// TIA Portal V17 export
// export: Created 2025-03-05T07:59:29.2018149Z, ExportSetting WithDefaults, DisplayName Totally Integrated Automation Portal, DisplayVersion V17 Update 8, DisplayName TIA Portal Openness, DisplayVersion V17 Update 8, DisplayName TIA Portal Version Control Interface, DisplayVersion V17, DisplayName SINAMICS Startdrive Advanced, DisplayVersion V17 SP2, DisplayName SINAMICS Startdrive G110M, G120, G120C, G120D, G120P, G115D, DisplayVersion V17 SP2, DisplayName SINAMICS Startdrive G130, G150, S120, S150, SINAMICS MV, S210, DisplayVersion V17 SP2, DisplayName STEP 7 Professional, DisplayVersion V17 Update 8, DisplayName SINUMERIK ONE STEP 7 Toolbox, DisplayVersion V17 Update 12, DisplayName SINUMERIK 840D sl STEP 7 Toolbox, DisplayVersion V17 Update 12, DisplayName STEP 7 Safety, DisplayVersion V17 Update 6, DisplayName WinCC Advanced, DisplayVersion V17 Update 8
FUNCTION_BLOCK "FB301_CHANNEL_READ_AXES_POSITIONS"   // FB301, LAD
{ S7_Optimized_Access := 'FALSE' }
AUTHOR : ETXETAR
VERSION : 1.0
// stored: AutoNumber false, IsIECCheckEnabled false, SetENOAutomatically false, UDAEnableTagReadback false
   VAR_INPUT
      NUMBER_AXES_GROUP_1 : Int;   // MAX. VALUE 8 / NUMBER AXES GROUP 1, MAX=8
      NUMBER_AXES_GROUP_2 : Int;   // MAX. VALUE 7 / NUMBER AXES GROUP 2, MAX=8
      NUMBER_AXES_GROUP_3 : Int;   // MAX. VALUE 7 / NUMBER AXES GROUP 3, MAX=4
   END_VAR
   VAR_OUTPUT
      ALARM : Bool;   // ALARM
      AXIS_POSITION_1 : DWord;   // AXIS POSITION 1
      AXIS_POSITION_2 : DWord;   // AXIS POSITION 2
      AXIS_POSITION_3 : DWord;   // AXIS POSITION 3
      AXIS_POSITION_4 : DWord;   // AXIS POSITION 4
      AXIS_POSITION_5 : DWord;   // AXIS POSITION 5
      AXIS_POSITION_6 : DWord;   // AXIS POSITION 6
      AXIS_POSITION_7 : DWord;   // AXIS POSITION 7
      AXIS_POSITION_8 : DWord;   // AXIS POSITION 8
      AXIS_POSITION_9 : DWord;   // AXIS POSITION 9
      AXIS_POSITION_10 : DWord;   // AXIS POSITION 10
      AXIS_POSITION_11 : DWord;   // AXIS POSITION 11
      AXIS_POSITION_12 : DWord;   // AXIS POSITION 12
      AXIS_POSITION_13 : DWord;   // AXIS POSITION 13
      AXIS_POSITION_14 : DWord;   // AXIS POSITION 14
      AXIS_POSITION_15 : DWord;   // AXIS POSITION 15
      AXIS_POSITION_16 : DWord;   // AXIS POSITION 16
      AXIS_POSITION_17 : DWord;   // AXIS POSITION 17
      AXIS_POSITION_18 : DWord;   // AXIS POSITION 18
      AXIS_POSITION_19 : DWord;   // AXIS POSITION 19
      AXIS_POSITION_20 : DWord;   // AXIS POSITION 20
   END_VAR
   VAR DB_SPECIFIC
      readDB { S7_SetPoint := 'True'} : "READ_AXES_POSITIONS_CH";
   END_VAR
   VAR
      FB2_Instance_1 { S7_SetPoint := 'True'} : "LBP_ReadVar";
      FB2_Instance_2 { S7_SetPoint := 'True'} : "LBP_ReadVar";
      FB2_Instance_3 { S7_SetPoint := 'True'} : "LBP_ReadVar";
   END_VAR
   VAR DB_SPECIFIC
      FAULT_COUNTER { S7_SetPoint := 'True'} : CTU_INT;
   END_VAR
   VAR_TEMP
      DB_NUMBER : DInt;   // DB NUMBER FOR ALARM AND HELP DECODING
      CHANNEL : UInt;   // CHANNEL NUMBER MAX. NUMBER=10
      FAULT : Bool;   // FAULT
      COUNT_ERRORS : Int;   // COUNT_ERRORS
   END_VAR
   VAR_TEMP   // added for the SCL form of the ladder/FBD networks
      _w1 : Bool;
   END_VAR
BEGIN

NETWORK
TITLE = READ INSTANCE DB
      L     DINO;
      +     10#800000;
      T     #DB_NUMBER;
      L     DINO;
      L     10#300;
      -I;
      T     #CHANNEL;



REGION Network 2: FAULT / CHANNELS READING FAULT
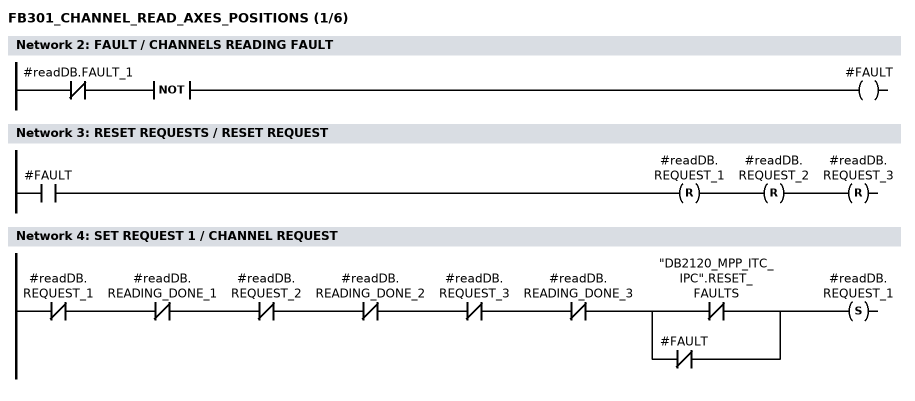
   RUNG wire#powerrail
      I_Contact( #readDB.FAULT_1 )
      Not()
      Coil( #FAULT )
   END_RUNG
   // the same network as SCL:
   #FAULT := NOT (NOT #readDB.FAULT_1);
END_REGION

REGION Network 3: RESET REQUESTS / RESET REQUEST
   RUNG wire#powerrail
      Contact( #FAULT )
      R_Coil( #readDB.REQUEST_1 )
      R_Coil( #readDB.REQUEST_2 )
      R_Coil( #readDB.REQUEST_3 )
   END_RUNG
   // the same network as SCL:
   IF #FAULT THEN
       #readDB.REQUEST_1 := FALSE;
       #readDB.REQUEST_2 := FALSE;
       #readDB.REQUEST_3 := FALSE;
   END_IF;
END_REGION

REGION Network 4: SET REQUEST 1 / CHANNEL REQUEST
   RUNG wire#powerrail
      I_Contact( #readDB.REQUEST_1 )
      I_Contact( #readDB.READING_DONE_1 )
      I_Contact( #readDB.REQUEST_2 )
      I_Contact( #readDB.READING_DONE_2 )
      I_Contact( #readDB.REQUEST_3 )
      I_Contact( #readDB.READING_DONE_3 )
      wire#w1
      I_Contact( "DB2120_MPP_ITC_IPC".RESET_FAULTS )
      wire#w2
      S_Coil( #readDB.REQUEST_1 )
   END_RUNG
   RUNG wire#w1
      I_Contact( #FAULT )
   END_RUNG wire#w2
   // the same network as SCL:
   IF NOT #readDB.REQUEST_1 AND NOT #readDB.READING_DONE_1 AND NOT #readDB.REQUEST_2 AND NOT #readDB.READING_DONE_2 AND NOT #readDB.REQUEST_3 AND NOT #readDB.READING_DONE_3 AND (NOT "DB2120_MPP_ITC_IPC".RESET_FAULTS OR NOT #FAULT) THEN
       #readDB.REQUEST_1 := TRUE;
   END_IF;
END_REGION

REGION Network 5: CALL FB2 GROUP 1 / READ AXES POSITIONS CHANNEL
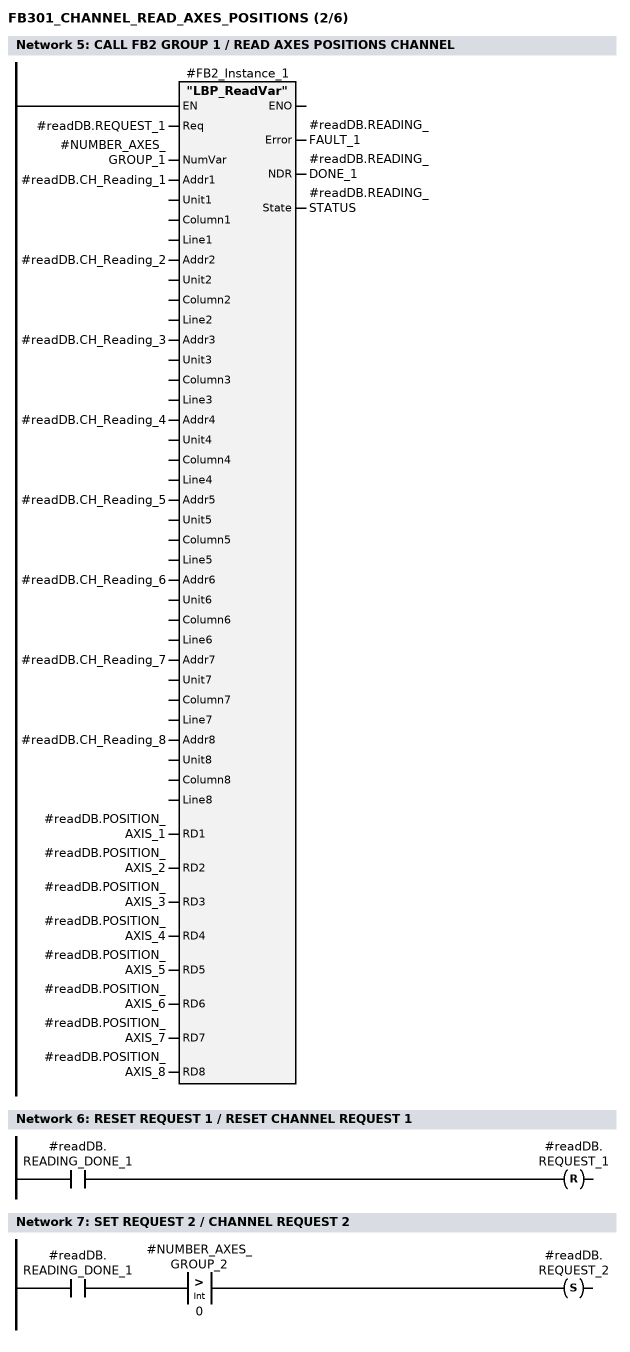
   RUNG wire#powerrail
      #FB2_Instance_1(Req := #readDB.REQUEST_1, NumVar := #NUMBER_AXES_GROUP_1, Addr1 := #readDB.CH_Reading_1, Unit1 :=, Column1 :=, Line1 :=, Addr2 := #readDB.CH_Reading_2, Unit2 :=, Column2 :=, Line2 :=, Addr3 := #readDB.CH_Reading_3, Unit3 :=, Column3 :=, Line3 :=, Addr4 := #readDB.CH_Reading_4, Unit4 :=, Column4 :=, Line4 :=, Addr5 := #readDB.CH_Reading_5, Unit5 :=, Column5 :=, Line5 :=, Addr6 := #readDB.CH_Reading_6, Unit6 :=, Column6 :=, Line6 :=, Addr7 := #readDB.CH_Reading_7, Unit7 :=, Column7 :=, Line7 :=, Addr8 := #readDB.CH_Reading_8, Unit8 :=, Column8 :=, Line8 :=, RD1 := #readDB.POSITION_AXIS_1, RD2 := #readDB.POSITION_AXIS_2, RD3 := #readDB.POSITION_AXIS_3, RD4 := #readDB.POSITION_AXIS_4, RD5 := #readDB.POSITION_AXIS_5, RD6 := #readDB.POSITION_AXIS_6, RD7 := #readDB.POSITION_AXIS_7, RD8 := #readDB.POSITION_AXIS_8, Error => #readDB.READING_FAULT_1, NDR => #readDB.READING_DONE_1, State => #readDB.READING_STATUS)
   END_RUNG
   // the same network as SCL:
   #FB2_Instance_1(Req := #readDB.REQUEST_1,   // "LBP_ReadVar"
                   NumVar := #NUMBER_AXES_GROUP_1,
                   Addr1 := #readDB.CH_Reading_1,
                   Addr2 := #readDB.CH_Reading_2,
                   Addr3 := #readDB.CH_Reading_3,
                   Addr4 := #readDB.CH_Reading_4,
                   Addr5 := #readDB.CH_Reading_5,
                   Addr6 := #readDB.CH_Reading_6,
                   Addr7 := #readDB.CH_Reading_7,
                   Addr8 := #readDB.CH_Reading_8,
                   RD1 := #readDB.POSITION_AXIS_1,
                   RD2 := #readDB.POSITION_AXIS_2,
                   RD3 := #readDB.POSITION_AXIS_3,
                   RD4 := #readDB.POSITION_AXIS_4,
                   RD5 := #readDB.POSITION_AXIS_5,
                   RD6 := #readDB.POSITION_AXIS_6,
                   RD7 := #readDB.POSITION_AXIS_7,
                   RD8 := #readDB.POSITION_AXIS_8,
                   Error => #readDB.READING_FAULT_1,
                   NDR => #readDB.READING_DONE_1,
                   State => #readDB.READING_STATUS);
END_REGION

REGION Network 6: RESET REQUEST 1 / RESET CHANNEL REQUEST 1
   RUNG wire#powerrail
      Contact( #readDB.READING_DONE_1 )
      R_Coil( #readDB.REQUEST_1 )
   END_RUNG
   // the same network as SCL:
   IF #readDB.READING_DONE_1 THEN #readDB.REQUEST_1 := FALSE; END_IF;
END_REGION

REGION Network 7: SET REQUEST 2 / CHANNEL REQUEST 2
   RUNG wire#powerrail
      Contact( #readDB.READING_DONE_1 )
      { S7_Templates := "SrcType := Int" } GT_Contact(in1 := #NUMBER_AXES_GROUP_2, in2 := 0)
      S_Coil( #readDB.REQUEST_2 )
   END_RUNG
   // the same network as SCL:
   IF #readDB.READING_DONE_1 AND (#NUMBER_AXES_GROUP_2 > 0) THEN #readDB.REQUEST_2 := TRUE; END_IF;
END_REGION

REGION Network 8: CALL FB2 GROUP 2 / READ AXES POSITIONS CHANNEL
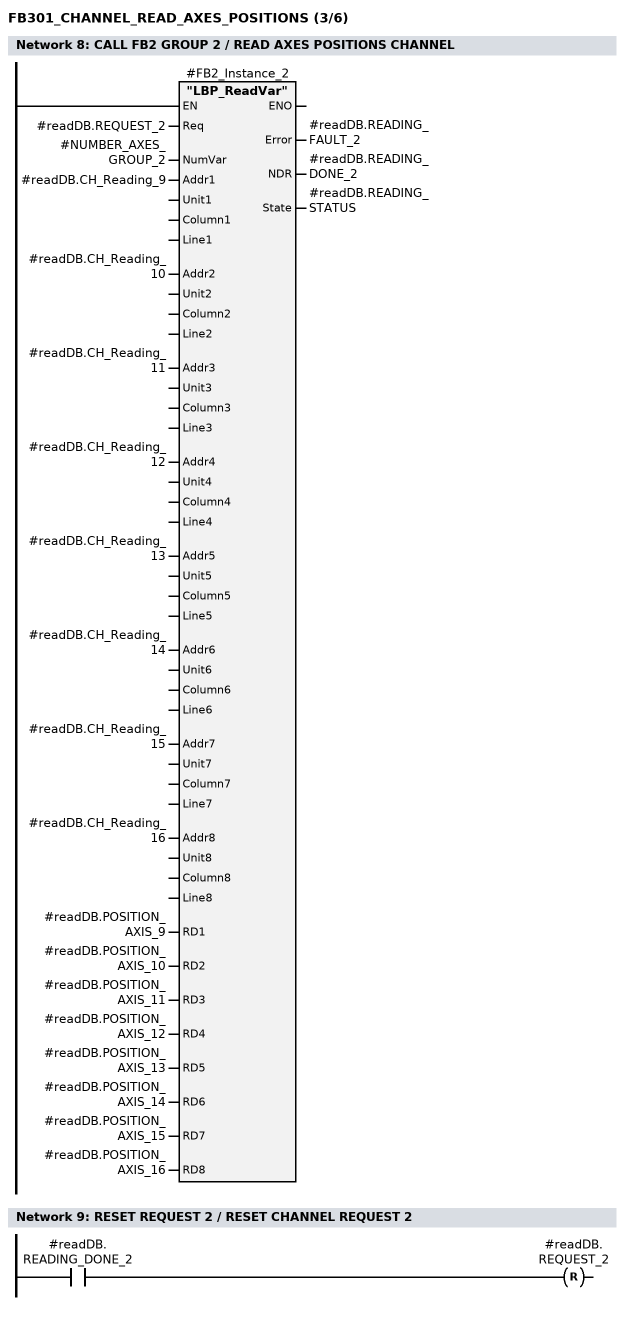
   RUNG wire#powerrail
      #FB2_Instance_2(Req := #readDB.REQUEST_2, NumVar := #NUMBER_AXES_GROUP_2, Addr1 := #readDB.CH_Reading_9, Unit1 :=, Column1 :=, Line1 :=, Addr2 := #readDB.CH_Reading_10, Unit2 :=, Column2 :=, Line2 :=, Addr3 := #readDB.CH_Reading_11, Unit3 :=, Column3 :=, Line3 :=, Addr4 := #readDB.CH_Reading_12, Unit4 :=, Column4 :=, Line4 :=, Addr5 := #readDB.CH_Reading_13, Unit5 :=, Column5 :=, Line5 :=, Addr6 := #readDB.CH_Reading_14, Unit6 :=, Column6 :=, Line6 :=, Addr7 := #readDB.CH_Reading_15, Unit7 :=, Column7 :=, Line7 :=, Addr8 := #readDB.CH_Reading_16, Unit8 :=, Column8 :=, Line8 :=, RD1 := #readDB.POSITION_AXIS_9, RD2 := #readDB.POSITION_AXIS_10, RD3 := #readDB.POSITION_AXIS_11, RD4 := #readDB.POSITION_AXIS_12, RD5 := #readDB.POSITION_AXIS_13, RD6 := #readDB.POSITION_AXIS_14, RD7 := #readDB.POSITION_AXIS_15, RD8 := #readDB.POSITION_AXIS_16, Error => #readDB.READING_FAULT_2, NDR => #readDB.READING_DONE_2, State => #readDB.READING_STATUS)
   END_RUNG
   // the same network as SCL:
   #FB2_Instance_2(Req := #readDB.REQUEST_2,   // "LBP_ReadVar"
                   NumVar := #NUMBER_AXES_GROUP_2,
                   Addr1 := #readDB.CH_Reading_9,
                   Addr2 := #readDB.CH_Reading_10,
                   Addr3 := #readDB.CH_Reading_11,
                   Addr4 := #readDB.CH_Reading_12,
                   Addr5 := #readDB.CH_Reading_13,
                   Addr6 := #readDB.CH_Reading_14,
                   Addr7 := #readDB.CH_Reading_15,
                   Addr8 := #readDB.CH_Reading_16,
                   RD1 := #readDB.POSITION_AXIS_9,
                   RD2 := #readDB.POSITION_AXIS_10,
                   RD3 := #readDB.POSITION_AXIS_11,
                   RD4 := #readDB.POSITION_AXIS_12,
                   RD5 := #readDB.POSITION_AXIS_13,
                   RD6 := #readDB.POSITION_AXIS_14,
                   RD7 := #readDB.POSITION_AXIS_15,
                   RD8 := #readDB.POSITION_AXIS_16,
                   Error => #readDB.READING_FAULT_2,
                   NDR => #readDB.READING_DONE_2,
                   State => #readDB.READING_STATUS);
END_REGION

REGION Network 9: RESET REQUEST 2 / RESET CHANNEL REQUEST 2
   RUNG wire#powerrail
      Contact( #readDB.READING_DONE_2 )
      R_Coil( #readDB.REQUEST_2 )
   END_RUNG
   // the same network as SCL:
   IF #readDB.READING_DONE_2 THEN #readDB.REQUEST_2 := FALSE; END_IF;
END_REGION

REGION Network 10: SET REQUEST 3 / RESET CHANNEL REQUEST 2
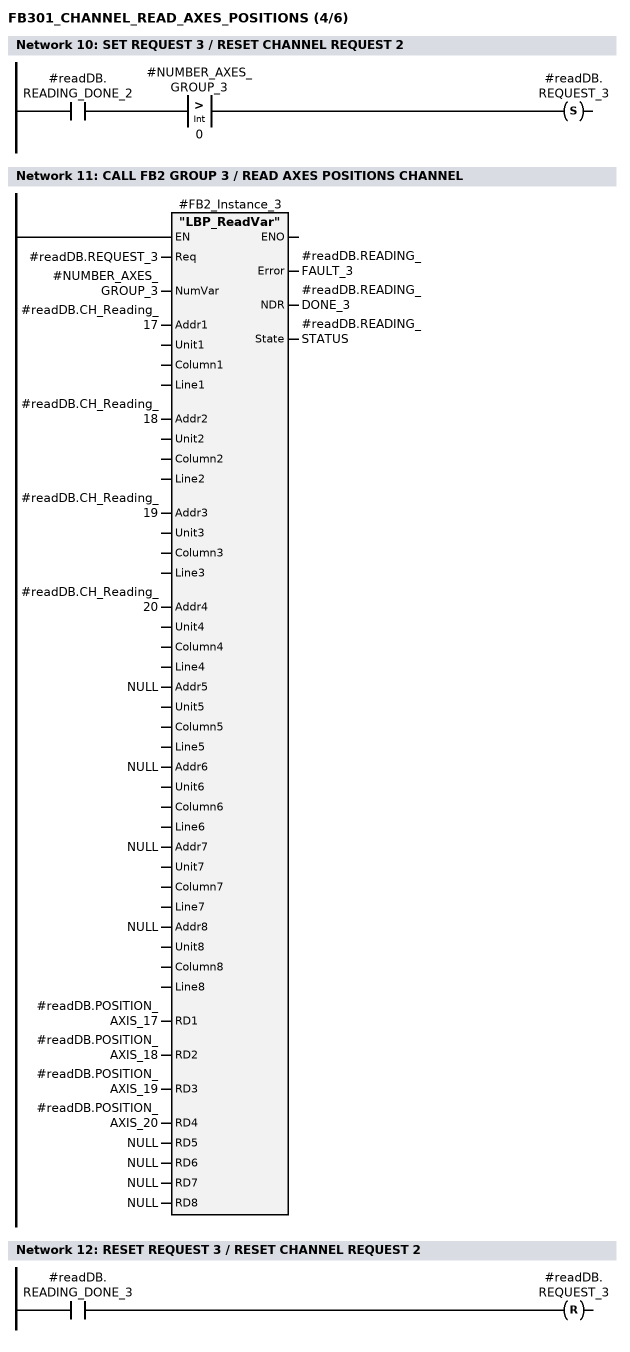
   RUNG wire#powerrail
      Contact( #readDB.READING_DONE_2 )
      { S7_Templates := "SrcType := Int" } GT_Contact(in1 := #NUMBER_AXES_GROUP_3, in2 := 0)
      S_Coil( #readDB.REQUEST_3 )
   END_RUNG
   // the same network as SCL:
   IF #readDB.READING_DONE_2 AND (#NUMBER_AXES_GROUP_3 > 0) THEN #readDB.REQUEST_3 := TRUE; END_IF;
END_REGION

REGION Network 11: CALL FB2 GROUP 3 / READ AXES POSITIONS CHANNEL
   RUNG wire#powerrail
      #FB2_Instance_3(Req := #readDB.REQUEST_3, NumVar := #NUMBER_AXES_GROUP_3, Addr1 := #readDB.CH_Reading_17, Unit1 :=, Column1 :=, Line1 :=, Addr2 := #readDB.CH_Reading_18, Unit2 :=, Column2 :=, Line2 :=, Addr3 := #readDB.CH_Reading_19, Unit3 :=, Column3 :=, Line3 :=, Addr4 := #readDB.CH_Reading_20, Unit4 :=, Column4 :=, Line4 :=, Addr5 := NULL, Unit5 :=, Column5 :=, Line5 :=, Addr6 := NULL, Unit6 :=, Column6 :=, Line6 :=, Addr7 := NULL, Unit7 :=, Column7 :=, Line7 :=, Addr8 := NULL, Unit8 :=, Column8 :=, Line8 :=, RD1 := #readDB.POSITION_AXIS_17, RD2 := #readDB.POSITION_AXIS_18, RD3 := #readDB.POSITION_AXIS_19, RD4 := #readDB.POSITION_AXIS_20, RD5 := NULL, RD6 := NULL, RD7 := NULL, RD8 := NULL, Error => #readDB.READING_FAULT_3, NDR => #readDB.READING_DONE_3, State => #readDB.READING_STATUS)
   END_RUNG
   // the same network as SCL:
   #FB2_Instance_3(Req := #readDB.REQUEST_3,   // "LBP_ReadVar"
                   NumVar := #NUMBER_AXES_GROUP_3,
                   Addr1 := #readDB.CH_Reading_17,
                   Addr2 := #readDB.CH_Reading_18,
                   Addr3 := #readDB.CH_Reading_19,
                   Addr4 := #readDB.CH_Reading_20,
                   Addr5 := NULL,
                   Addr6 := NULL,
                   Addr7 := NULL,
                   Addr8 := NULL,
                   RD1 := #readDB.POSITION_AXIS_17,
                   RD2 := #readDB.POSITION_AXIS_18,
                   RD3 := #readDB.POSITION_AXIS_19,
                   RD4 := #readDB.POSITION_AXIS_20,
                   RD5 := NULL,
                   RD6 := NULL,
                   RD7 := NULL,
                   RD8 := NULL,
                   Error => #readDB.READING_FAULT_3,
                   NDR => #readDB.READING_DONE_3,
                   State => #readDB.READING_STATUS);
END_REGION

REGION Network 12: RESET REQUEST 3 / RESET CHANNEL REQUEST 2
   RUNG wire#powerrail
      Contact( #readDB.READING_DONE_3 )
      R_Coil( #readDB.REQUEST_3 )
   END_RUNG
   // the same network as SCL:
   IF #readDB.READING_DONE_3 THEN #readDB.REQUEST_3 := FALSE; END_IF;
END_REGION

REGION Network 13: MOVE POSITIONS / AXES POSITIONS
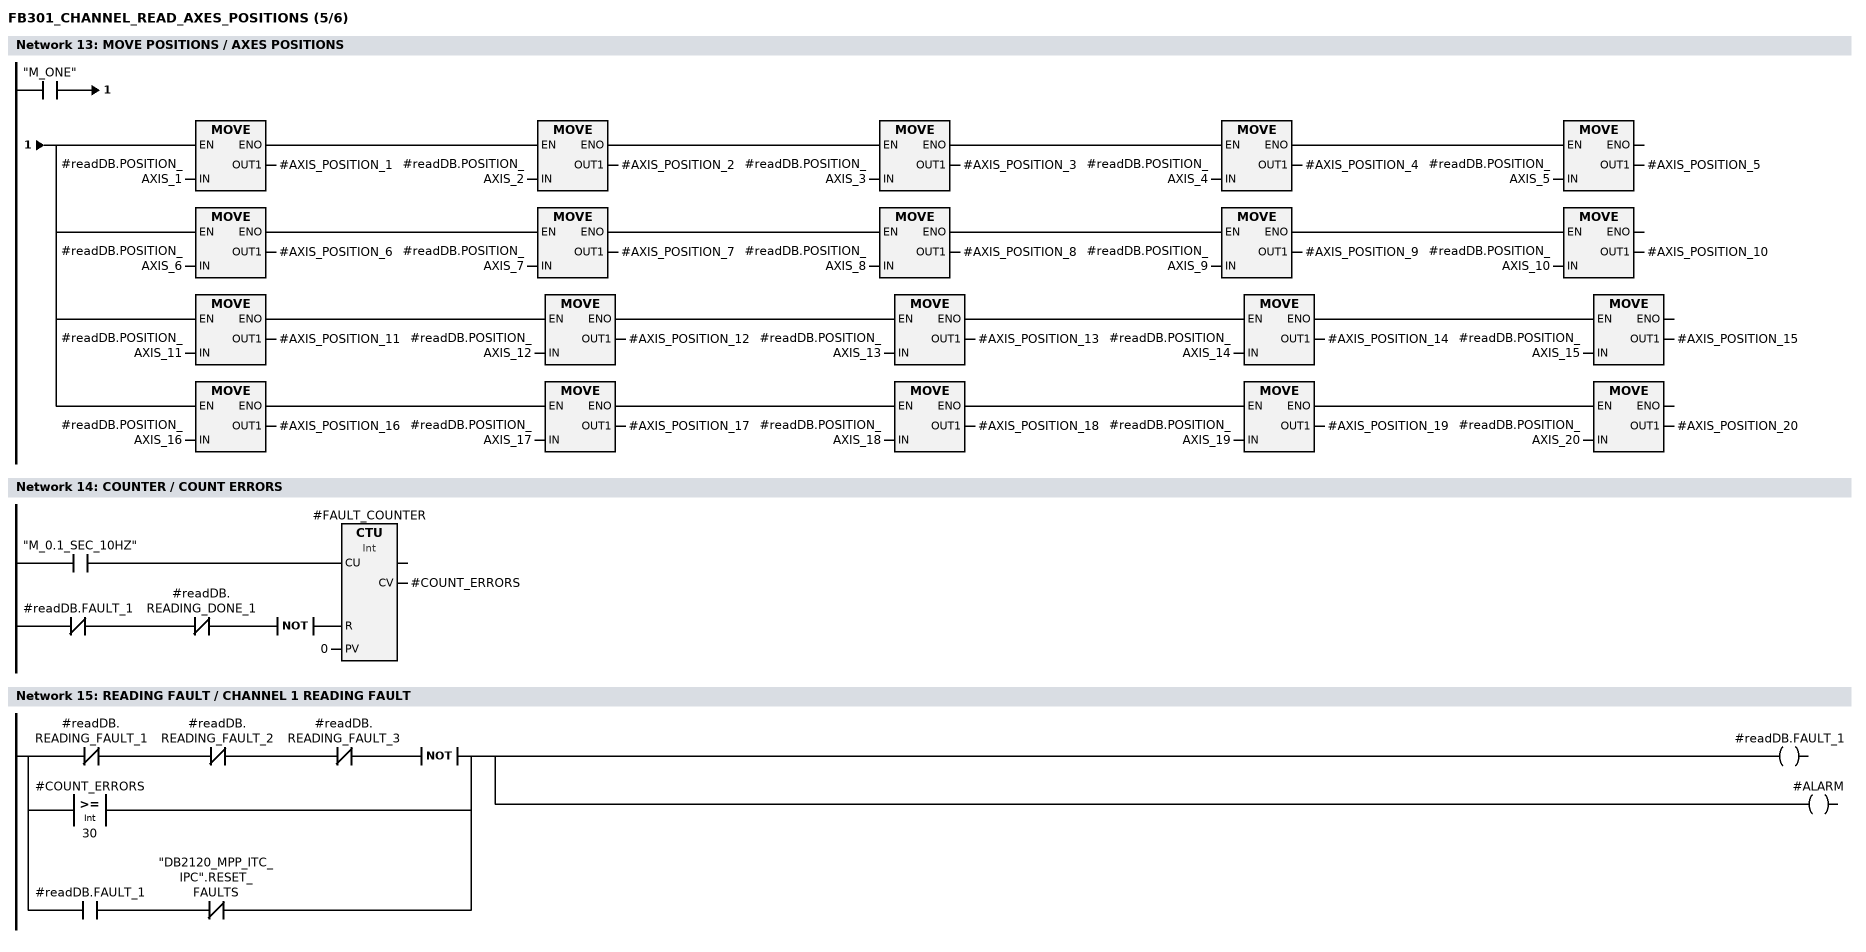
   RUNG wire#powerrail
      Contact( "M_ONE" )
      wire#w1
      { S7_GenerateENO := "TRUE" } Move(in := #readDB.POSITION_AXIS_1, out1 => #AXIS_POSITION_1)
      { S7_GenerateENO := "TRUE" } Move(in := #readDB.POSITION_AXIS_2, out1 => #AXIS_POSITION_2)
      { S7_GenerateENO := "TRUE" } Move(in := #readDB.POSITION_AXIS_3, out1 => #AXIS_POSITION_3)
      { S7_GenerateENO := "TRUE" } Move(in := #readDB.POSITION_AXIS_4, out1 => #AXIS_POSITION_4)
      { S7_GenerateENO := "TRUE" } Move(in := #readDB.POSITION_AXIS_5, out1 => #AXIS_POSITION_5)
   END_RUNG
   RUNG wire#w1
      { S7_GenerateENO := "TRUE" } Move(in := #readDB.POSITION_AXIS_6, out1 => #AXIS_POSITION_6)
      { S7_GenerateENO := "TRUE" } Move(in := #readDB.POSITION_AXIS_7, out1 => #AXIS_POSITION_7)
      { S7_GenerateENO := "TRUE" } Move(in := #readDB.POSITION_AXIS_8, out1 => #AXIS_POSITION_8)
      { S7_GenerateENO := "TRUE" } Move(in := #readDB.POSITION_AXIS_9, out1 => #AXIS_POSITION_9)
      { S7_GenerateENO := "TRUE" } Move(in := #readDB.POSITION_AXIS_10, out1 => #AXIS_POSITION_10)
   END_RUNG
   RUNG wire#w1
      { S7_GenerateENO := "TRUE" } Move(in := #readDB.POSITION_AXIS_11, out1 => #AXIS_POSITION_11)
      { S7_GenerateENO := "TRUE" } Move(in := #readDB.POSITION_AXIS_12, out1 => #AXIS_POSITION_12)
      { S7_GenerateENO := "TRUE" } Move(in := #readDB.POSITION_AXIS_13, out1 => #AXIS_POSITION_13)
      { S7_GenerateENO := "TRUE" } Move(in := #readDB.POSITION_AXIS_14, out1 => #AXIS_POSITION_14)
      { S7_GenerateENO := "TRUE" } Move(in := #readDB.POSITION_AXIS_15, out1 => #AXIS_POSITION_15)
   END_RUNG
   RUNG wire#w1
      { S7_GenerateENO := "TRUE" } Move(in := #readDB.POSITION_AXIS_16, out1 => #AXIS_POSITION_16)
      { S7_GenerateENO := "TRUE" } Move(in := #readDB.POSITION_AXIS_17, out1 => #AXIS_POSITION_17)
      { S7_GenerateENO := "TRUE" } Move(in := #readDB.POSITION_AXIS_18, out1 => #AXIS_POSITION_18)
      { S7_GenerateENO := "TRUE" } Move(in := #readDB.POSITION_AXIS_19, out1 => #AXIS_POSITION_19)
      { S7_GenerateENO := "TRUE" } Move(in := #readDB.POSITION_AXIS_20, out1 => #AXIS_POSITION_20)
   END_RUNG
   // the same network as SCL:
   // ENO of a box is taken as its EN; it also drops when the box reports an error
   IF "M_ONE" THEN
       #AXIS_POSITION_1 := #readDB.POSITION_AXIS_1;
       #AXIS_POSITION_2 := #readDB.POSITION_AXIS_2;
       #AXIS_POSITION_3 := #readDB.POSITION_AXIS_3;
       #AXIS_POSITION_4 := #readDB.POSITION_AXIS_4;
       #AXIS_POSITION_5 := #readDB.POSITION_AXIS_5;
       #AXIS_POSITION_6 := #readDB.POSITION_AXIS_6;
       #AXIS_POSITION_7 := #readDB.POSITION_AXIS_7;
       #AXIS_POSITION_8 := #readDB.POSITION_AXIS_8;
       #AXIS_POSITION_9 := #readDB.POSITION_AXIS_9;
       #AXIS_POSITION_10 := #readDB.POSITION_AXIS_10;
       #AXIS_POSITION_11 := #readDB.POSITION_AXIS_11;
       #AXIS_POSITION_12 := #readDB.POSITION_AXIS_12;
       #AXIS_POSITION_13 := #readDB.POSITION_AXIS_13;
       #AXIS_POSITION_14 := #readDB.POSITION_AXIS_14;
       #AXIS_POSITION_15 := #readDB.POSITION_AXIS_15;
       #AXIS_POSITION_16 := #readDB.POSITION_AXIS_16;
       #AXIS_POSITION_17 := #readDB.POSITION_AXIS_17;
       #AXIS_POSITION_18 := #readDB.POSITION_AXIS_18;
       #AXIS_POSITION_19 := #readDB.POSITION_AXIS_19;
       #AXIS_POSITION_20 := #readDB.POSITION_AXIS_20;
   END_IF;
END_REGION

REGION Network 14: COUNTER / COUNT ERRORS
   RUNG wire#powerrail
      Contact( "M_0.1_SEC_10HZ" )
      { S7_Templates := "value_type := Int" } #FAULT_COUNTER.CTU(r := wire#w1, pv := 0, cv => #COUNT_ERRORS)
   END_RUNG
   RUNG wire#powerrail
      I_Contact( #readDB.FAULT_1 )
      I_Contact( #readDB.READING_DONE_1 )
      Not()
   END_RUNG wire#w1
   // the same network as SCL:
   #FAULT_COUNTER(CU := "M_0.1_SEC_10HZ",   // CTU
                  R := NOT (NOT #readDB.FAULT_1 AND NOT #readDB.READING_DONE_1),
                  PV := 0,
                  CV => #COUNT_ERRORS);
END_REGION

REGION Network 15: READING FAULT / CHANNEL 1 READING FAULT
   RUNG wire#powerrail
      I_Contact( #readDB.READING_FAULT_1 )
      I_Contact( #readDB.READING_FAULT_2 )
      I_Contact( #readDB.READING_FAULT_3 )
      Not()
      wire#w1
      Coil( #readDB.FAULT_1 )
   END_RUNG
   RUNG wire#powerrail
      { S7_Templates := "SrcType := Int" } GE_Contact(in1 := #COUNT_ERRORS, in2 := 30)
   END_RUNG wire#w1
   RUNG wire#powerrail
      Contact( #readDB.FAULT_1 )
      I_Contact( "DB2120_MPP_ITC_IPC".RESET_FAULTS )
   END_RUNG wire#w1
   RUNG wire#w1
      Coil( #ALARM )
   END_RUNG
   // the same network as SCL:
   #readDB.FAULT_1 := NOT (NOT #readDB.READING_FAULT_1 AND NOT #readDB.READING_FAULT_2 AND NOT #readDB.READING_FAULT_3) OR (#COUNT_ERRORS >= 30) OR (#readDB.FAULT_1 AND NOT "DB2120_MPP_ITC_IPC".RESET_FAULTS);
   #ALARM := #readDB.FAULT_1;
END_REGION

REGION Network 16: IMMEDIATE STOP AND STOP END OF CYCLE ALARMS / IMMEDIATE STOP ALARMS
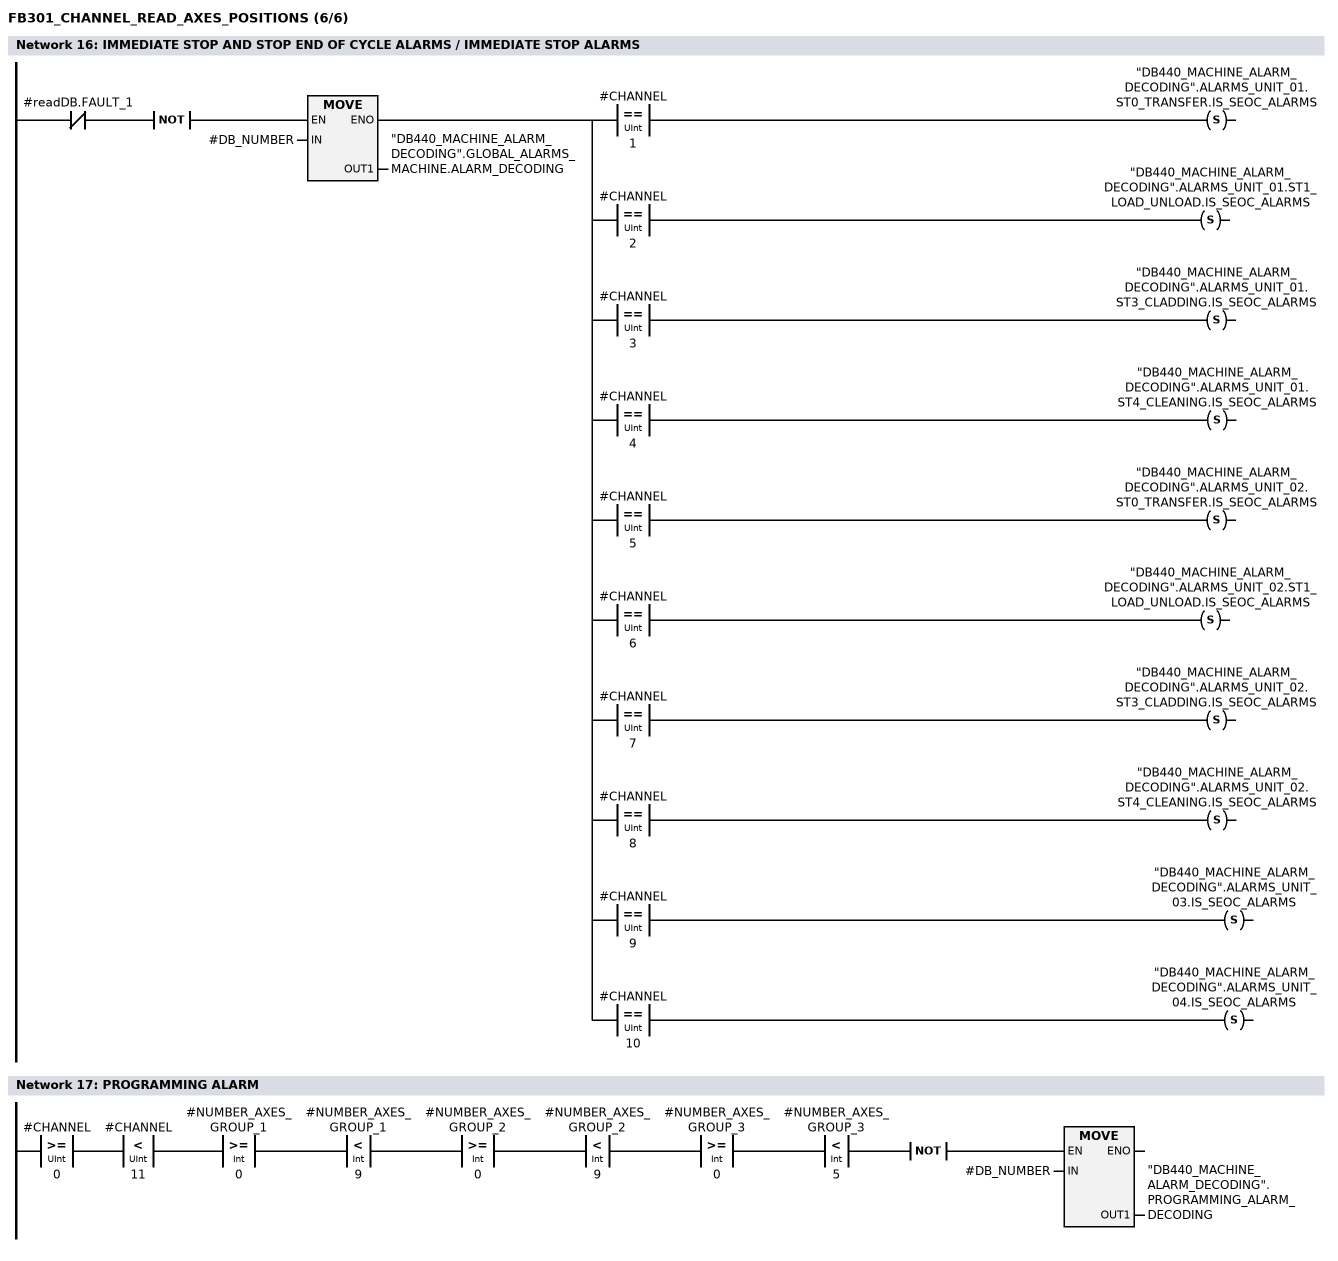
   RUNG wire#powerrail
      I_Contact( #readDB.FAULT_1 )
      Not()
      { S7_GenerateENO := "TRUE" } Move(in := #DB_NUMBER, out1 => "DB440_MACHINE_ALARM_DECODING".GLOBAL_ALARMS_MACHINE.ALARM_DECODING)
      wire#w1
      { S7_Templates := "SrcType := UInt" } EQ_Contact(in1 := #CHANNEL, in2 := 1)
      S_Coil( "DB440_MACHINE_ALARM_DECODING".ALARMS_UNIT_01.ST0_TRANSFER.IS_SEOC_ALARMS )
   END_RUNG
   RUNG wire#w1
      { S7_Templates := "SrcType := UInt" } EQ_Contact(in1 := #CHANNEL, in2 := 2)
      S_Coil( "DB440_MACHINE_ALARM_DECODING".ALARMS_UNIT_01.ST1_LOAD_UNLOAD.IS_SEOC_ALARMS )
   END_RUNG
   RUNG wire#w1
      { S7_Templates := "SrcType := UInt" } EQ_Contact(in1 := #CHANNEL, in2 := 3)
      S_Coil( "DB440_MACHINE_ALARM_DECODING".ALARMS_UNIT_01.ST3_CLADDING.IS_SEOC_ALARMS )
   END_RUNG
   RUNG wire#w1
      { S7_Templates := "SrcType := UInt" } EQ_Contact(in1 := #CHANNEL, in2 := 4)
      S_Coil( "DB440_MACHINE_ALARM_DECODING".ALARMS_UNIT_01.ST4_CLEANING.IS_SEOC_ALARMS )
   END_RUNG
   RUNG wire#w1
      { S7_Templates := "SrcType := UInt" } EQ_Contact(in1 := #CHANNEL, in2 := 5)
      S_Coil( "DB440_MACHINE_ALARM_DECODING".ALARMS_UNIT_02.ST0_TRANSFER.IS_SEOC_ALARMS )
   END_RUNG
   RUNG wire#w1
      { S7_Templates := "SrcType := UInt" } EQ_Contact(in1 := #CHANNEL, in2 := 6)
      S_Coil( "DB440_MACHINE_ALARM_DECODING".ALARMS_UNIT_02.ST1_LOAD_UNLOAD.IS_SEOC_ALARMS )
   END_RUNG
   RUNG wire#w1
      { S7_Templates := "SrcType := UInt" } EQ_Contact(in1 := #CHANNEL, in2 := 7)
      S_Coil( "DB440_MACHINE_ALARM_DECODING".ALARMS_UNIT_02.ST3_CLADDING.IS_SEOC_ALARMS )
   END_RUNG
   RUNG wire#w1
      { S7_Templates := "SrcType := UInt" } EQ_Contact(in1 := #CHANNEL, in2 := 8)
      S_Coil( "DB440_MACHINE_ALARM_DECODING".ALARMS_UNIT_02.ST4_CLEANING.IS_SEOC_ALARMS )
   END_RUNG
   RUNG wire#w1
      { S7_Templates := "SrcType := UInt" } EQ_Contact(in1 := #CHANNEL, in2 := 9)
      S_Coil( "DB440_MACHINE_ALARM_DECODING".ALARMS_UNIT_03.IS_SEOC_ALARMS )
   END_RUNG
   RUNG wire#w1
      { S7_Templates := "SrcType := UInt" } EQ_Contact(in1 := #CHANNEL, in2 := 10)
      S_Coil( "DB440_MACHINE_ALARM_DECODING".ALARMS_UNIT_04.IS_SEOC_ALARMS )
   END_RUNG
   // the same network as SCL:
   // ENO of a box is taken as its EN; it also drops when the box reports an error
   #_w1 := NOT (NOT #readDB.FAULT_1);
   IF #_w1 THEN "DB440_MACHINE_ALARM_DECODING".GLOBAL_ALARMS_MACHINE.ALARM_DECODING := #DB_NUMBER; END_IF;
   IF #_w1 AND (#CHANNEL = 1) THEN
       "DB440_MACHINE_ALARM_DECODING".ALARMS_UNIT_01.ST0_TRANSFER.IS_SEOC_ALARMS := TRUE;
   END_IF;
   IF #_w1 AND (#CHANNEL = 2) THEN
       "DB440_MACHINE_ALARM_DECODING".ALARMS_UNIT_01.ST1_LOAD_UNLOAD.IS_SEOC_ALARMS := TRUE;
   END_IF;
   IF #_w1 AND (#CHANNEL = 3) THEN
       "DB440_MACHINE_ALARM_DECODING".ALARMS_UNIT_01.ST3_CLADDING.IS_SEOC_ALARMS := TRUE;
   END_IF;
   IF #_w1 AND (#CHANNEL = 4) THEN
       "DB440_MACHINE_ALARM_DECODING".ALARMS_UNIT_01.ST4_CLEANING.IS_SEOC_ALARMS := TRUE;
   END_IF;
   IF #_w1 AND (#CHANNEL = 5) THEN
       "DB440_MACHINE_ALARM_DECODING".ALARMS_UNIT_02.ST0_TRANSFER.IS_SEOC_ALARMS := TRUE;
   END_IF;
   IF #_w1 AND (#CHANNEL = 6) THEN
       "DB440_MACHINE_ALARM_DECODING".ALARMS_UNIT_02.ST1_LOAD_UNLOAD.IS_SEOC_ALARMS := TRUE;
   END_IF;
   IF #_w1 AND (#CHANNEL = 7) THEN
       "DB440_MACHINE_ALARM_DECODING".ALARMS_UNIT_02.ST3_CLADDING.IS_SEOC_ALARMS := TRUE;
   END_IF;
   IF #_w1 AND (#CHANNEL = 8) THEN
       "DB440_MACHINE_ALARM_DECODING".ALARMS_UNIT_02.ST4_CLEANING.IS_SEOC_ALARMS := TRUE;
   END_IF;
   IF #_w1 AND (#CHANNEL = 9) THEN
       "DB440_MACHINE_ALARM_DECODING".ALARMS_UNIT_03.IS_SEOC_ALARMS := TRUE;
   END_IF;
   IF #_w1 AND (#CHANNEL = 10) THEN
       "DB440_MACHINE_ALARM_DECODING".ALARMS_UNIT_04.IS_SEOC_ALARMS := TRUE;
   END_IF;
END_REGION

REGION Network 17: PROGRAMMING ALARM
   RUNG wire#powerrail
      { S7_Templates := "SrcType := UInt" } GE_Contact(in1 := #CHANNEL, in2 := 0)
      { S7_Templates := "SrcType := UInt" } LT_Contact(in1 := #CHANNEL, in2 := 11)
      { S7_Templates := "SrcType := Int" } GE_Contact(in1 := #NUMBER_AXES_GROUP_1, in2 := 0)
      { S7_Templates := "SrcType := Int" } LT_Contact(in1 := #NUMBER_AXES_GROUP_1, in2 := 9)
      { S7_Templates := "SrcType := Int" } GE_Contact(in1 := #NUMBER_AXES_GROUP_2, in2 := 0)
      { S7_Templates := "SrcType := Int" } LT_Contact(in1 := #NUMBER_AXES_GROUP_2, in2 := 9)
      { S7_Templates := "SrcType := Int" } GE_Contact(in1 := #NUMBER_AXES_GROUP_3, in2 := 0)
      { S7_Templates := "SrcType := Int" } LT_Contact(in1 := #NUMBER_AXES_GROUP_3, in2 := 5)
      Not()
      Move(in := #DB_NUMBER, out1 => "DB440_MACHINE_ALARM_DECODING".PROGRAMMING_ALARM_DECODING)
   END_RUNG
   // the same network as SCL:
   IF NOT ((#CHANNEL >= 0) AND (#CHANNEL < 11) AND (#NUMBER_AXES_GROUP_1 >= 0) AND (#NUMBER_AXES_GROUP_1 < 9) AND (#NUMBER_AXES_GROUP_2 >= 0) AND (#NUMBER_AXES_GROUP_2 < 9) AND (#NUMBER_AXES_GROUP_3 >= 0) AND (#NUMBER_AXES_GROUP_3 < 5)) THEN
       "DB440_MACHINE_ALARM_DECODING".PROGRAMMING_ALARM_DECODING := #DB_NUMBER;
   END_IF;
END_REGION
END_FUNCTION_BLOCK
